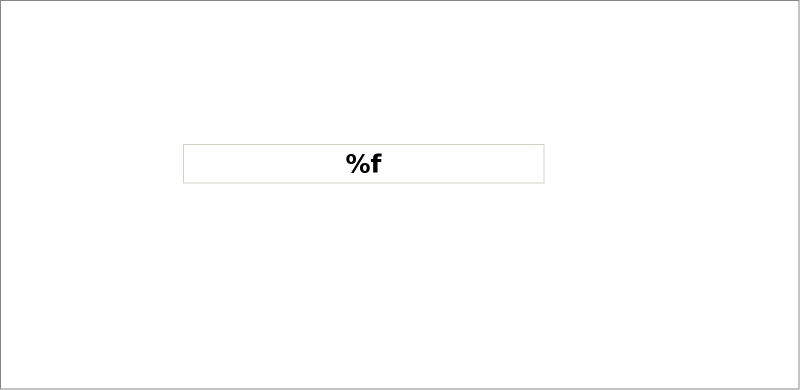
VISUALIZATION VisuEncoderInput  // 800x390
    Textfield (183,144 361x39), "%f", text variable: GVL_DevManual.fbManualControler.pDevEncoder^.nOutPosition
END_VISUALIZATION

(* stored: Version 1.1.0.1, ProductVersion 3.1.4024.5
   Visu VisuEncoderInput: Id {9f88dfcc-1ec2-4c14-8b61-63c3ccc32078} *)
